ABB RobotStudio station: parte0_clase.rspag

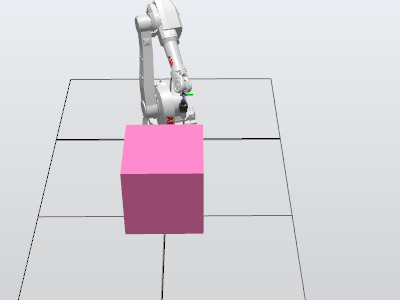
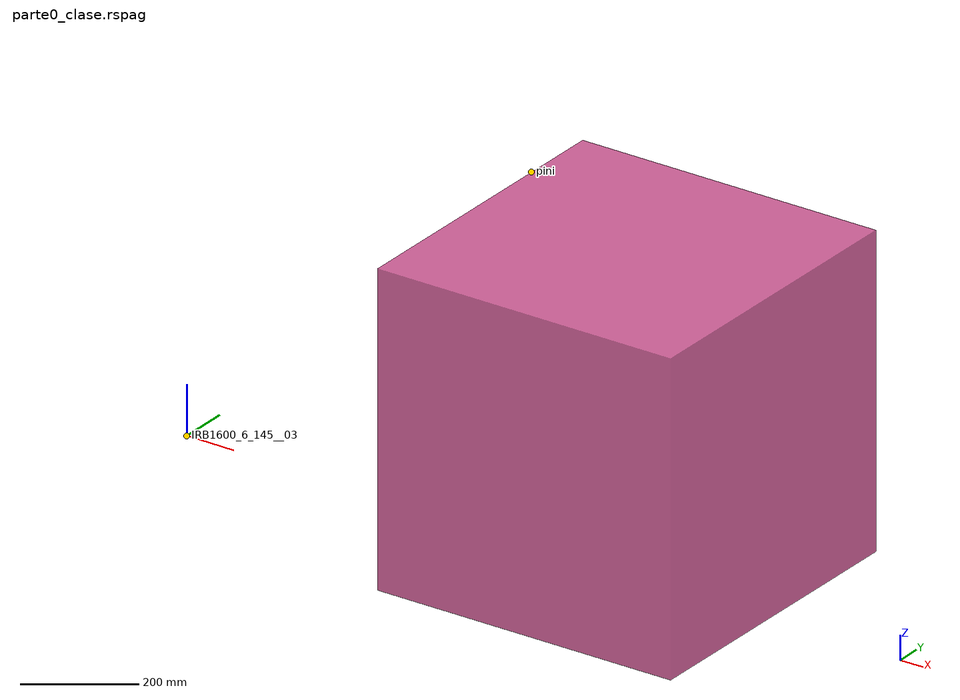
[picture v1: parts stored in the station drawn from their meshes, with robot base, taught points and paths (robot models come from the ABB library and are not in the file)]
--- station ---
Station parte0 (saved by RobotStudio 24.1.10713.1)
Controller Controlador3
  mechanical unit ROB_1: IRB1600_6_145__03, 6 joints, base frame (0, 0, 0) mm
Layout (positions relative to the parent item):
  - IRB1600_6_145__03 [mechanism, from %ABB.RobotStudio.Models.IRB1600%\IRB1600_6_145_G_03.rslib] at (0, 0, 0) mm; joint values [0.326, -0.2862, 0.8219, -0.4788, 0.4423, 0.699] (rad or m)
  - MyTool [mechanism, from Training Objects\myTool.rslib] at (483.67, 150, 800.53) mm, rotated rx -180 ry 38 rz -180 deg
  - Pieza_1 [part], size 600 x 600 x 600 mm
Attachment: MyTool is attached to IRB1600_6_145__03 / Link6
Targets, tools, work objects and paths stored in the station and not in the controller backup, written as RAPID:
! task T_ROB1
MODULE Module1
  PROC Path_10()
    MoveL pini,v1000,z100,MyTool\WObj:=wobj0;
  ENDPROC
ENDMODULE


--- Backups/Controlador3/RAPID/TASK1/PROGMOD/CalibData.mod ---
MODULE CalibData
    PERS tooldata MyTool:=[TRUE,[[31.792631019,0,229.638935148],[0.945518576,0,0.325568154,0]],[1,[0,0,1],[1,0,0,0],0,0,0]];
ENDMODULE

--- Backups/Controlador3/RAPID/TASK1/PROGMOD/Module1.mod ---
MODULE Module1
        CONST robtarget pini:=[[600,150,600],[0,0,1,0],[0,0,0,0],[9E+09,9E+09,9E+09,9E+09,9E+09,9E+09]];

    PROC main()
       Senoide pini, 100,40;
    ENDPROC
    PROC Senoide(robtarget pInicial, num amplx, num amplY)
        CONST num nPuntos :=50;
        VAR robtarget pVector{nPuntos};
        VAR robtarget pAux;
        VAR num xDesp;
        VAR num yDesp;
        !el movimiento en x es posicion inicial en x +2x
        !regla  3
        ! rela de 3 en grados
        !var robtarget pFinal := Offs(pInicial,2*amplx,0,0) ;
        MoveL pini,v1000,z100,MyTool\WObj:=wobj0;
        FOR i FROM 1 TO nPuntos DO
            !si queremos que el punto inicial cuente como parte de los puntos
            !2 opciones
            !1) Dentro del primer bucle,una condicion que haga que cuando i valga uno pvector{i} = pini(ideal si hacemos el camino inverso )
            !2) reducir el número de puntos en 1
         xDesp:= (i/nPuntos) * 2*amplx;
         yDesp:= Sin ((i/nPuntos)*360)* amplY;
        ! pAux:= Offs (pini, xDesp, yDesp , 0);
           !pVector{i}:= pAux;
         pVector{i}:= pini;
         pVector{i}.trans.x:= pVector{i}.trans.x + xDesp;
         pVector{i}.trans.y:= pVector{i}.trans.y + yDesp;


        ENDFOR
        FOR i FROM 1 TO nPuntos DO
            MoveL pVector{i},v100,z50,MyTool\WObj:=wobj0;
        ENDFOR
        MoveL pInicial,v100,z100,MyTool\WObj:=wobj0;


    ENDPROC
ENDMODULE
